Staubli VAL3: mnuMotionMenu.pgx

program mnuMotionMenu()
  local bool LbBackup
  local num nKey
begin
  //header begin
  // PROGRAM mnuMotionMenu()
  //
  // runs the menu to select various MOTION functions
  //
  // incoming parms:  none
  // outgoing parms:  none
  // called from:  pgm main()
  //
  //  initial release KN
  //  Release 3:  added F3 Button call to pgm <something>
  //  /per Blue Technik quote K01c, Work Request K01-1
  //header end
  //
  // start continuous loop, end by menu command or teach pendant command
  // on user command, jump to other subroutines for action
  //
  LbBackup=false
  do
    //nIdxMotionMenu=271
    call display(nIdxMotionMenu,nKey)
    // verify selection
    switch nKey
      // ESC key aborts & returns immediately
      case 255
        return
      break
      // Motion Menu:  F1 Button, go to Target Point menu for move & adjust functions
      case 271
        call mnuMoveTargPnt()
      break
      // Motion Menu:  F4 Button, Move to PARK position
      case 274
        call movToPark()
      break
      // Motion Menu:  F6 Button, Move to PARK TOP position
      case 276
        call movToParkTop()
      break
      // F8 Button, backup to Main Menu
      case 278
        LbBackup=true
      break
      // any other key press
      default
        cls()
        popUpMsg("BAD SELECTION...Press OK")
      break
    endSwitch
  until (false or (LbBackup==true))
  // done
end
